FUNCTION_BLOCK FB_ModeSelect
VAR_INPUT
	bControlBox : BOOL;
END_VAR
VAR_OUTPUT
END_VAR
VAR
	fbModeVisu : FB_ModeVisu;
	fbMode : I_Mode := fbModeVisu;
	fbModeCBox: FB_ModeCBox;
END_VAR

IF NOT (bControlBox) THEN
	
fbMode := fbModeVisu;
	IF NOT (HMI.stVisuParam.bOn) THEN
			fbMode.OFF(TRUE);
			fbMode.Auto(FALSE);
			fbMode.Manual(FALSE);
		
	ELSIF (HMI.stVisuParam.bOn) AND NOT (HMI.stVisuParam.bAuto) THEN
			fbMode.OFF(FALSE);
			fbMode.Auto(FALSE);
			fbMode.Manual(TRUE);
		
	ELSIF (HMI.stVisuParam.bOn) AND (HMI.stVisuParam.bAuto) THEN
			fbMode.OFF(FALSE);
			fbMode.Auto(TRUE);
			fbMode.Manual(FALSE);
		
	ELSE
			fbMode.OFF(FALSE);
			fbMode.Auto(FALSE);
			fbMode.Manual(FALSE);
		
	END_IF
	
ELSE
	
	fbMode := fbModeCBox;
	IF NOT (Input.stBoxParam.bAuto) AND NOT(Input.stBoxParam.bManual) THEN
			fbMode.OFF(TRUE);
			fbMode.Auto(FALSE);
			fbMode.Manual(FALSE);
		
	ELSIF NOT (Input.stBoxParam.bAuto) AND Input.stBoxParam.bManual THEN
			fbMode.OFF(FALSE);
			fbMode.Auto(FALSE);
			fbMode.Manual(TRUE);
		
	ELSIF NOT (Input.stBoxParam.bManual) AND Input.stBoxParam.bAuto THEN
			fbMode.OFF(FALSE);
			fbMode.Auto(TRUE);
			fbMode.Manual(FALSE);
		
	ELSE
			fbMode.OFF(FALSE);
			fbMode.Auto(FALSE);
			fbMode.Manual(FALSE);
		
	END_IF
	
END_IF

END_FUNCTION_BLOCK

(* stored: Version 1.1.0.1, ProductVersion 3.1.4024.12
   POU FB_ModeSelect: Id {881f20d6-17e9-402b-80f4-efea5e3c2672}, SpecialFunc None *)
